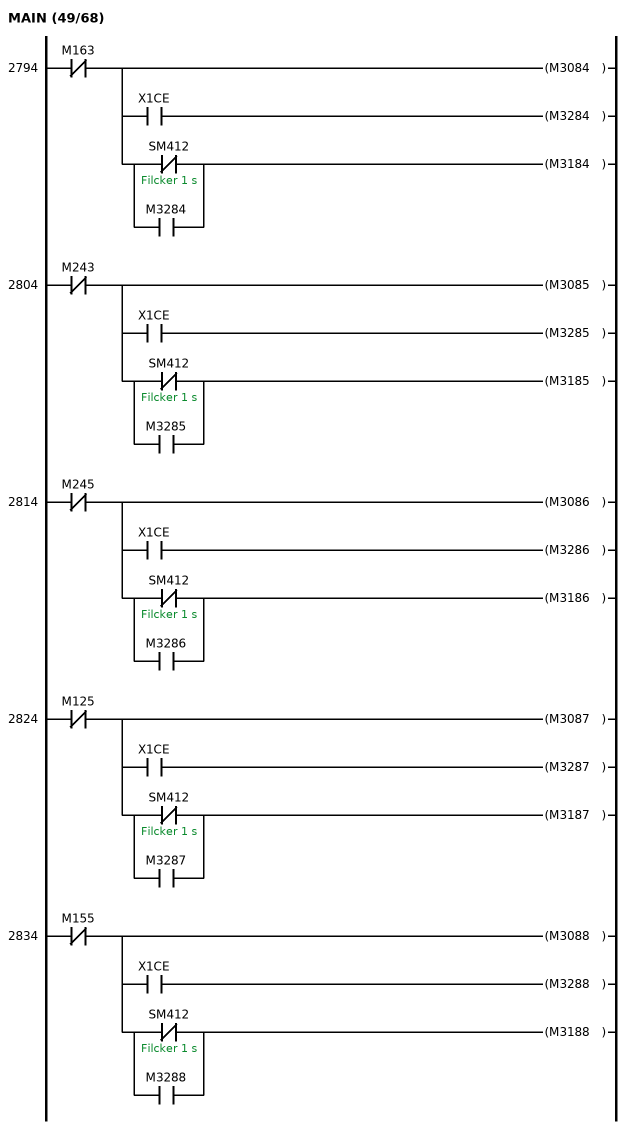
[picture p48: ladder of MAIN, rungs at steps 2794 to 2834]
2794  LDI     M163
      OUT     M3084
      MPS
      AND     X1CE
      OUT     M3284
      MPP
      LDI     SM412  ; Filcker 1 s
      OR      M3284
      ANB
      OUT     M3184
2804  LDI     M243
      OUT     M3085
      MPS
      AND     X1CE
      OUT     M3285
      MPP
      LDI     SM412  ; Filcker 1 s
      OR      M3285
      ANB
      OUT     M3185
2814  LDI     M245
      OUT     M3086
      MPS
      AND     X1CE
      OUT     M3286
      MPP
      LDI     SM412  ; Filcker 1 s
      OR      M3286
      ANB
      OUT     M3186
2824  LDI     M125
      OUT     M3087
      MPS
      AND     X1CE
      OUT     M3287
      MPP
      LDI     SM412  ; Filcker 1 s
      OR      M3287
      ANB
      OUT     M3187
2834  LDI     M155
      OUT     M3088
      MPS
      AND     X1CE
      OUT     M3288
      MPP
      LDI     SM412  ; Filcker 1 s
      OR      M3288
      ANB
      OUT     M3188
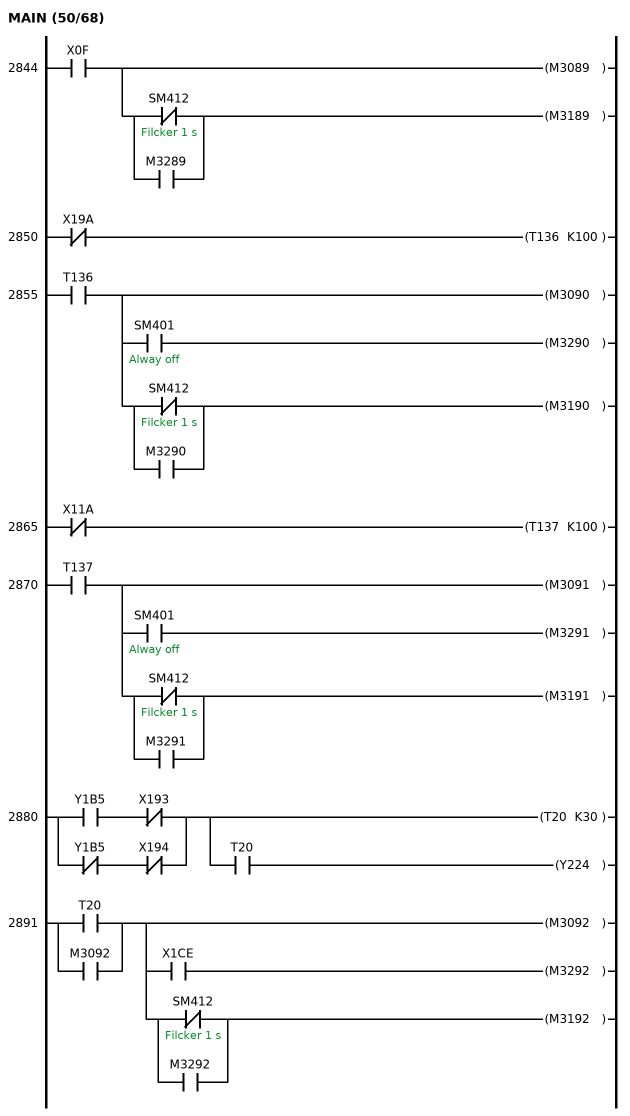
2844  LD      X0F
      OUT     M3089
      LDI     SM412  ; Filcker 1 s
      OR      M3289
      ANB
      OUT     M3189
2850  LDI     X19A
      OUT     T136 K100
2855  LD      T136
      OUT     M3090
      MPS
      AND     SM401  ; Alway off
      OUT     M3290
      MPP
      LDI     SM412  ; Filcker 1 s
      OR      M3290
      ANB
      OUT     M3190
2865  LDI     X11A
      OUT     T137 K100
2870  LD      T137
      OUT     M3091
      MPS
      AND     SM401  ; Alway off
      OUT     M3291
      MPP
      LDI     SM412  ; Filcker 1 s
      OR      M3291
      ANB
      OUT     M3191
2880  LD      Y1B5
      ANI     X193
      LDI     Y1B5
      ANI     X194
      ORB
      OUT     T20 K30
      AND     T20
      OUT     Y224
2891  LD      T20
      OR      M3092
      OUT     M3092
      MPS
      AND     X1CE
      OUT     M3292
      MPP
      LDI     SM412  ; Filcker 1 s
      OR      M3292
      ANB
      OUT     M3192
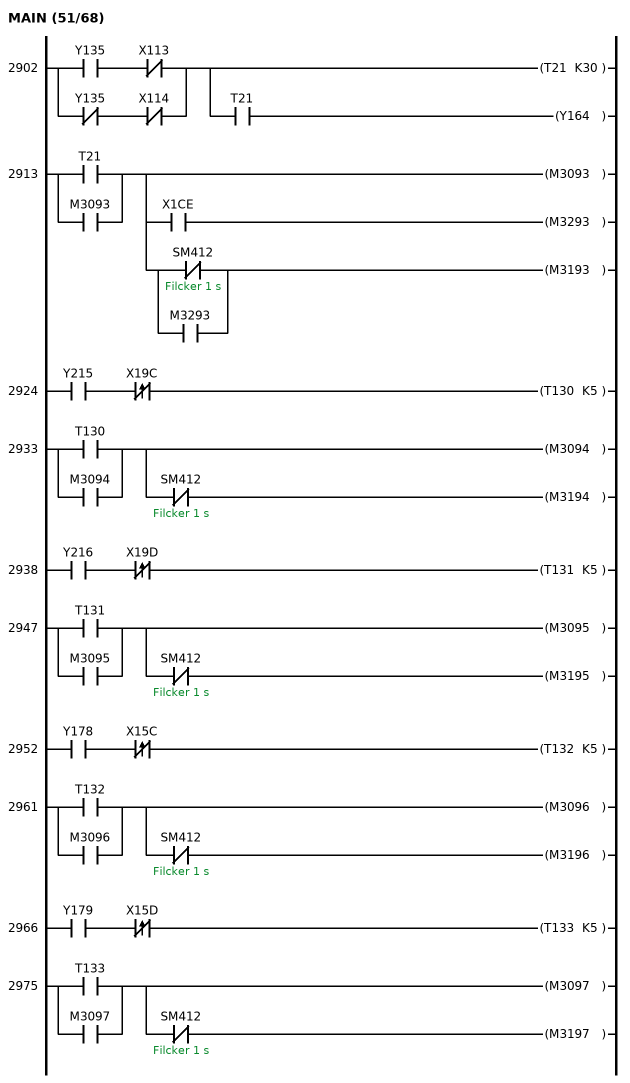
2902  LD      Y135
      ANI     X113
      LDI     Y135
      ANI     X114
      ORB
      OUT     T21 K30
      AND     T21
      OUT     Y164
2913  LD      T21
      OR      M3093
      OUT     M3093
      MPS
      AND     X1CE
      OUT     M3293
      MPP
      LDI     SM412  ; Filcker 1 s
      OR      M3293
      ANB
      OUT     M3193
2924  LD      Y215
      ANDPI   X19C
      OUT     T130 K5
2933  LD      T130
      OR      M3094
      OUT     M3094
      ANI     SM412  ; Filcker 1 s
      OUT     M3194
2938  LD      Y216
      ANDPI   X19D
      OUT     T131 K5
2947  LD      T131
      OR      M3095
      OUT     M3095
      ANI     SM412  ; Filcker 1 s
      OUT     M3195
2952  LD      Y178
      ANDPI   X15C
      OUT     T132 K5
2961  LD      T132
      OR      M3096
      OUT     M3096
      ANI     SM412  ; Filcker 1 s
      OUT     M3196
2966  LD      Y179
      ANDPI   X15D
      OUT     T133 K5
2975  LD      T133
      OR      M3097
      OUT     M3097
      ANI     SM412  ; Filcker 1 s
      OUT     M3197
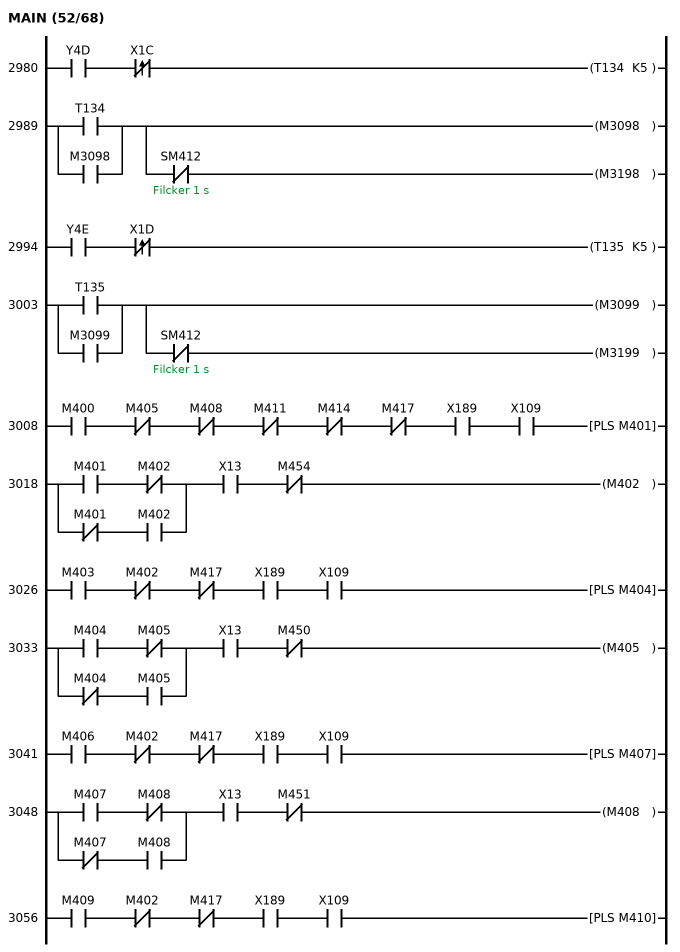
2980  LD      Y4D
      ANDPI   X1C
      OUT     T134 K5
2989  LD      T134
      OR      M3098
      OUT     M3098
      ANI     SM412  ; Filcker 1 s
      OUT     M3198
2994  LD      Y4E
      ANDPI   X1D
      OUT     T135 K5
3003  LD      T135
      OR      M3099
      OUT     M3099
      ANI     SM412  ; Filcker 1 s
      OUT     M3199
3008  LD      M400
      ANI     M405
      ANI     M408
      ANI     M411
      ANI     M414
      ANI     M417
      AND     X189
      AND     X109
      PLS     M401
3018  LD      M401
      ANI     M402
      LDI     M401
      AND     M402
      ORB
      AND     X13
      ANI     M454
      OUT     M402
3026  LD      M403
      ANI     M402
      ANI     M417
      AND     X189
      AND     X109
      PLS     M404
3033  LD      M404
      ANI     M405
      LDI     M404
      AND     M405
      ORB
      AND     X13
      ANI     M450
      OUT     M405
3041  LD      M406
      ANI     M402
      ANI     M417
      AND     X189
      AND     X109
      PLS     M407
3048  LD      M407
      ANI     M408
      LDI     M407
      AND     M408
      ORB
      AND     X13
      ANI     M451
      OUT     M408
3056  LD      M409
      ANI     M402
      ANI     M417
      AND     X189
      AND     X109
      PLS     M410
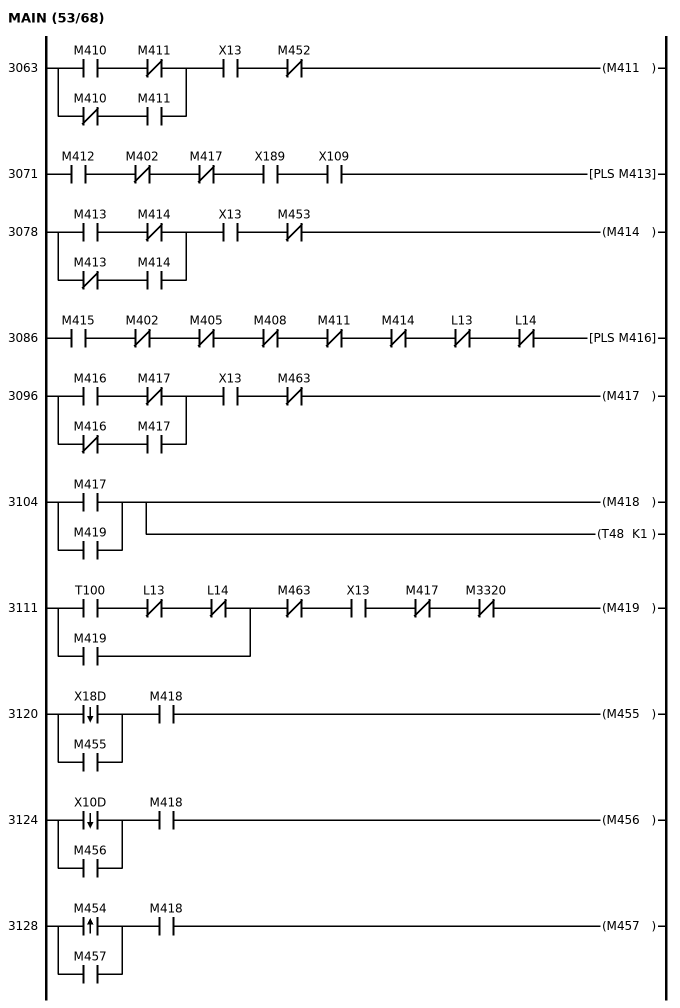
3063  LD      M410
      ANI     M411
      LDI     M410
      AND     M411
      ORB
      AND     X13
      ANI     M452
      OUT     M411
3071  LD      M412
      ANI     M402
      ANI     M417
      AND     X189
      AND     X109
      PLS     M413
3078  LD      M413
      ANI     M414
      LDI     M413
      AND     M414
      ORB
      AND     X13
      ANI     M453
      OUT     M414
3086  LD      M415
      ANI     M402
      ANI     M405
      ANI     M408
      ANI     M411
      ANI     M414
      ANI     L13
      ANI     L14
      PLS     M416
3096  LD      M416
      ANI     M417
      LDI     M416
      AND     M417
      ORB
      AND     X13
      ANI     M463
      OUT     M417
3104  LD      M417
      OR      M419
      OUT     M418
      OUT     T48 K1
3111  LD      T100
      ANI     L13
      ANI     L14
      OR      M419
      ANI     M463
      AND     X13
      ANI     M417
      ANI     M3320
      OUT     M419
3120  LDF     X18D
      OR      M455
      AND     M418
      OUT     M455
3124  LDF     X10D
      OR      M456
      AND     M418
      OUT     M456
3128  LDP     M454
      OR      M457
      AND     M418
      OUT     M457
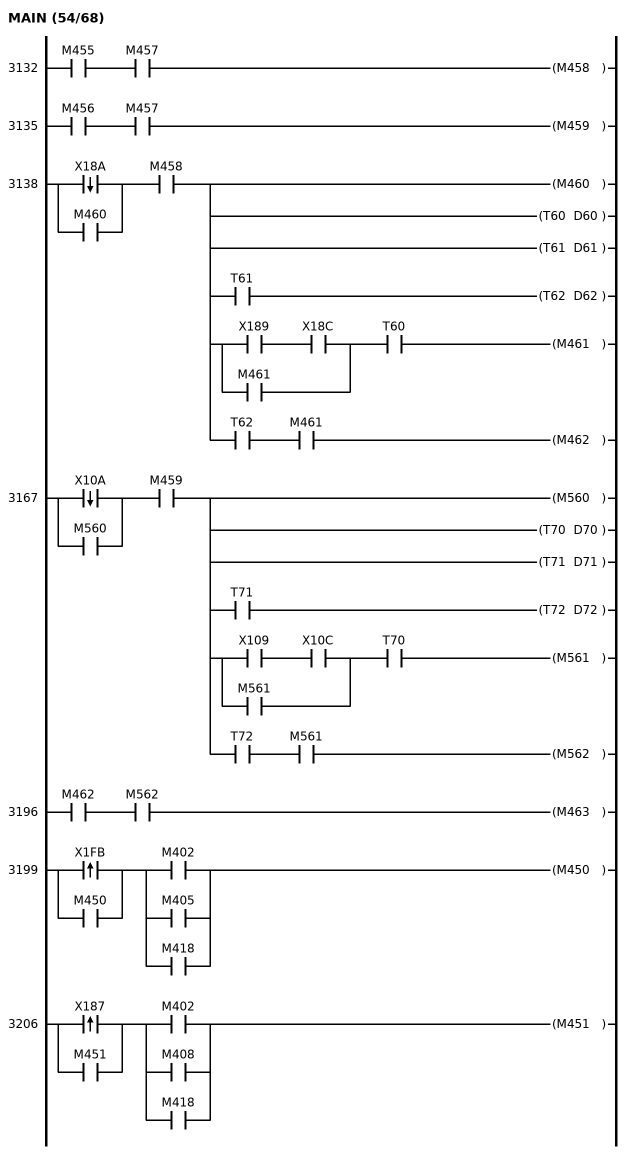
3132  LD      M455
      AND     M457
      OUT     M458
3135  LD      M456
      AND     M457
      OUT     M459
3138  LDF     X18A
      OR      M460
      AND     M458
      OUT     M460
      OUT     T60 D60
      OUT     T61 D61
      MPS
      AND     T61
      OUT     T62 D62
      MRD
      LD      X189
      AND     X18C
      OR      M461
      ANB
      AND     T60
      OUT     M461
      MPP
      AND     T62
      AND     M461
      OUT     M462
3167  LDF     X10A
      OR      M560
      AND     M459
      OUT     M560
      OUT     T70 D70
      OUT     T71 D71
      MPS
      AND     T71
      OUT     T72 D72
      MRD
      LD      X109
      AND     X10C
      OR      M561
      ANB
      AND     T70
      OUT     M561
      MPP
      AND     T72
      AND     M561
      OUT     M562
3196  LD      M462
      AND     M562
      OUT     M463
3199  LDP     X1FB
      OR      M450
      LD      M402
      OR      M405
      OR      M418
      ANB
      OUT     M450
3206  LDP     X187
      OR      M451
      LD      M402
      OR      M408
      OR      M418
      ANB
      OUT     M451
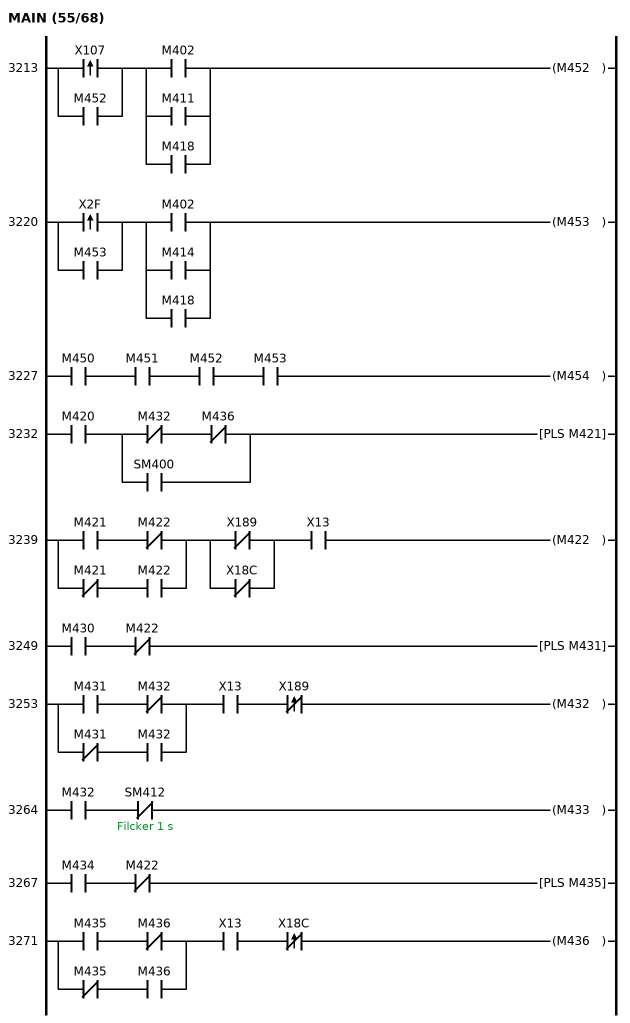
3213  LDP     X107
      OR      M452
      LD      M402
      OR      M411
      OR      M418
      ANB
      OUT     M452
3220  LDP     X2F
      OR      M453
      LD      M402
      OR      M414
      OR      M418
      ANB
      OUT     M453
3227  LD      M450
      AND     M451
      AND     M452
      AND     M453
      OUT     M454
3232  LD      M420
      LDI     M432
      ANI     M436
      OR      SM400
      ANB
      PLS     M421
3239  LD      M421
      ANI     M422
      LDI     M421
      AND     M422
      ORB
      LDI     X189
      ORI     X18C
      ANB
      AND     X13
      OUT     M422
3249  LD      M430
      ANI     M422
      PLS     M431
3253  LD      M431
      ANI     M432
      LDI     M431
      AND     M432
      ORB
      AND     X13
      ANDPI   X189
      OUT     M432
3264  LD      M432
      ANI     SM412  ; Filcker 1 s
      OUT     M433
3267  LD      M434
      ANI     M422
      PLS     M435
3271  LD      M435
      ANI     M436
      LDI     M435
      AND     M436
      ORB
      AND     X13
      ANDPI   X18C
      OUT     M436
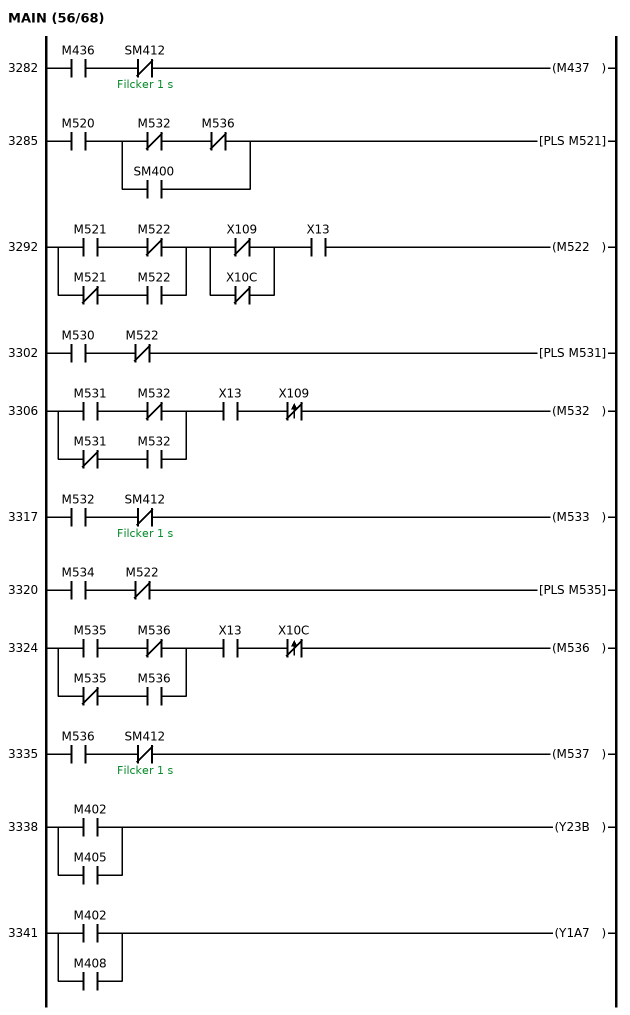
3282  LD      M436
      ANI     SM412  ; Filcker 1 s
      OUT     M437
3285  LD      M520
      LDI     M532
      ANI     M536
      OR      SM400
      ANB
      PLS     M521
3292  LD      M521
      ANI     M522
      LDI     M521
      AND     M522
      ORB
      LDI     X109
      ORI     X10C
      ANB
      AND     X13
      OUT     M522
3302  LD      M530
      ANI     M522
      PLS     M531
3306  LD      M531
      ANI     M532
      LDI     M531
      AND     M532
      ORB
      AND     X13
      ANDPI   X109
      OUT     M532
3317  LD      M532
      ANI     SM412  ; Filcker 1 s
      OUT     M533
3320  LD      M534
      ANI     M522
      PLS     M535
3324  LD      M535
      ANI     M536
      LDI     M535
      AND     M536
      ORB
      AND     X13
      ANDPI   X10C
      OUT     M536
3335  LD      M536
      ANI     SM412  ; Filcker 1 s
      OUT     M537
3338  LD      M402
      OR      M405
      OUT     Y23B
3341  LD      M402
      OR      M408
      OUT     Y1A7
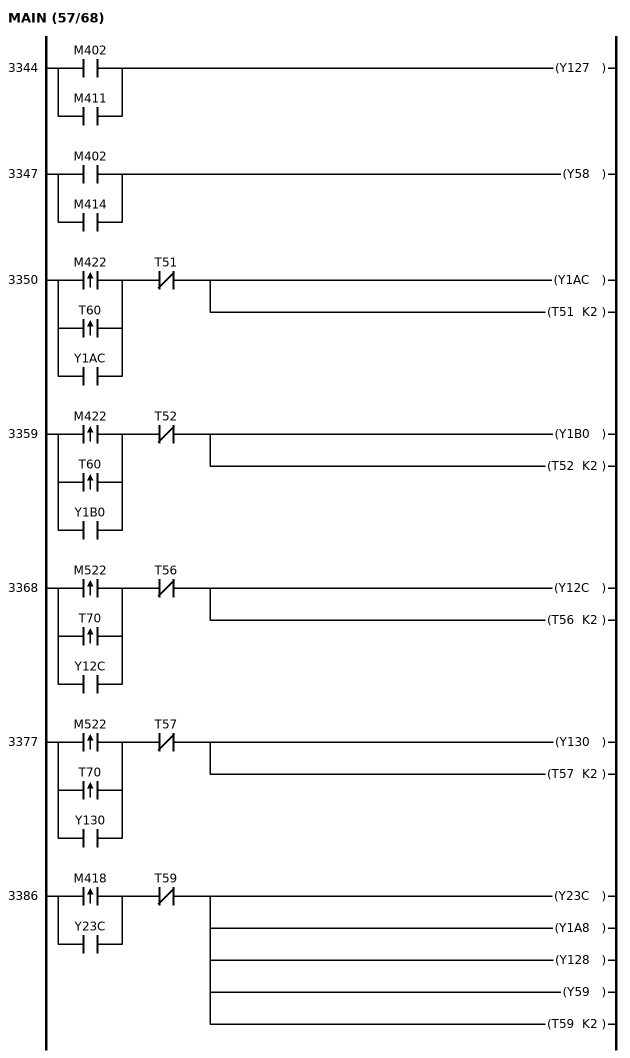
3344  LD      M402
      OR      M411
      OUT     Y127
3347  LD      M402
      OR      M414
      OUT     Y58
3350  LDP     M422
      ORP     T60
      OR      Y1AC
      ANI     T51
      OUT     Y1AC
      OUT     T51 K2
3359  LDP     M422
      ORP     T60
      OR      Y1B0
      ANI     T52
      OUT     Y1B0
      OUT     T52 K2
3368  LDP     M522
      ORP     T70
      OR      Y12C
      ANI     T56
      OUT     Y12C
      OUT     T56 K2
3377  LDP     M522
      ORP     T70
      OR      Y130
      ANI     T57
      OUT     Y130
      OUT     T57 K2
3386  LDP     M418
      OR      Y23C
      ANI     T59
      OUT     Y23C
      OUT     Y1A8
      OUT     Y128
      OUT     Y59
      OUT     T59 K2
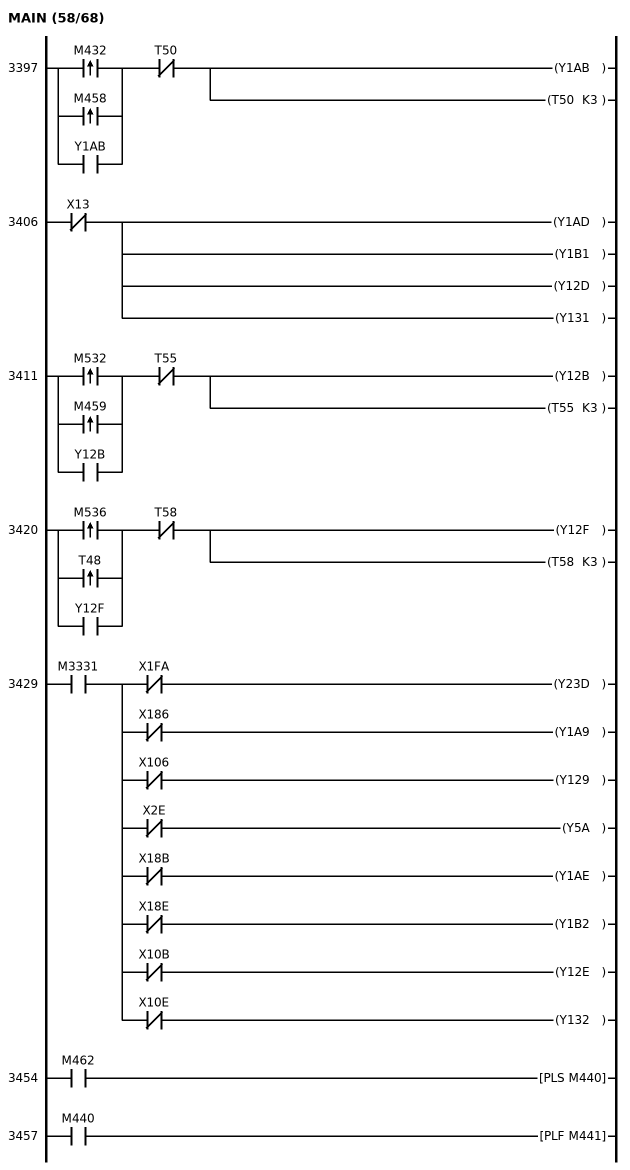
3397  LDP     M432
      ORP     M458
      OR      Y1AB
      ANI     T50
      OUT     Y1AB
      OUT     T50 K3
3406  LDI     X13
      OUT     Y1AD
      OUT     Y1B1
      OUT     Y12D
      OUT     Y131
3411  LDP     M532
      ORP     M459
      OR      Y12B
      ANI     T55
      OUT     Y12B
      OUT     T55 K3
3420  LDP     M536
      ORP     T48
      OR      Y12F
      ANI     T58
      OUT     Y12F
      OUT     T58 K3
3429  LD      M3331
      MPS
      ANI     X1FA
      OUT     Y23D
      MRD
      ANI     X186
      OUT     Y1A9
      MRD
      ANI     X106
      OUT     Y129
      MRD
      ANI     X2E
      OUT     Y5A
      MRD
      ANI     X18B
      OUT     Y1AE
      MRD
      ANI     X18E
      OUT     Y1B2
      MRD
      ANI     X10B
      OUT     Y12E
      MPP
      ANI     X10E
      OUT     Y132
3454  LD      M462
      PLS     M440
3457  LD      M440
      PLF     M441
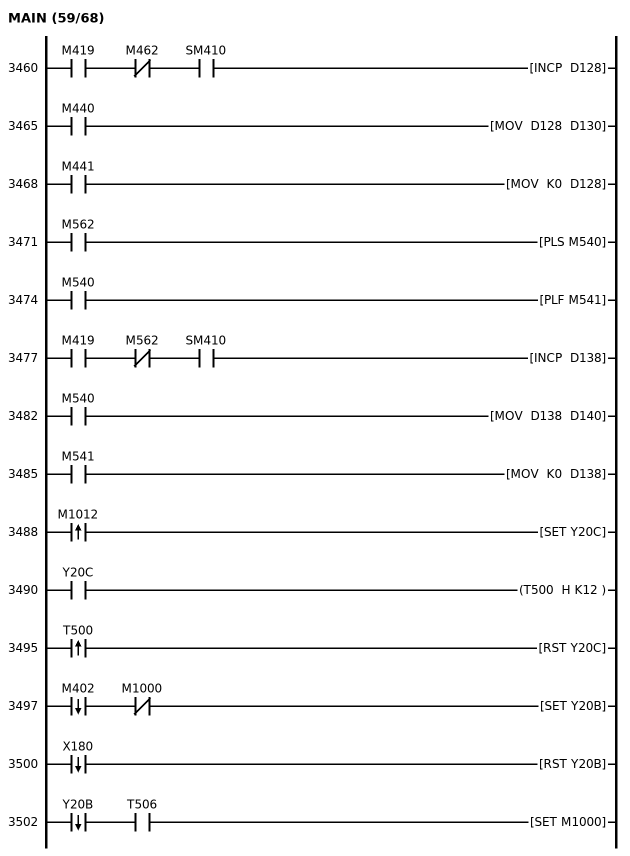
3460  LD      M419
      ANI     M462
      AND     SM410
      INCP    D128
3465  LD      M440
      MOV     D128 D130
3468  LD      M441
      MOV     K0 D128
3471  LD      M562
      PLS     M540
3474  LD      M540
      PLF     M541
3477  LD      M419
      ANI     M562
      AND     SM410
      INCP    D138
3482  LD      M540
      MOV     D138 D140
3485  LD      M541
      MOV     K0 D138
3488  LDP     M1012
      SET     Y20C
3490  LD      Y20C
      OUTH    T500 K12
3495  LDP     T500
      RST     Y20C
3497  LDF     M402
      ANI     M1000
      SET     Y20B
3500  LDF     X180
      RST     Y20B
3502  LDF     Y20B
      AND     T506
      SET     M1000
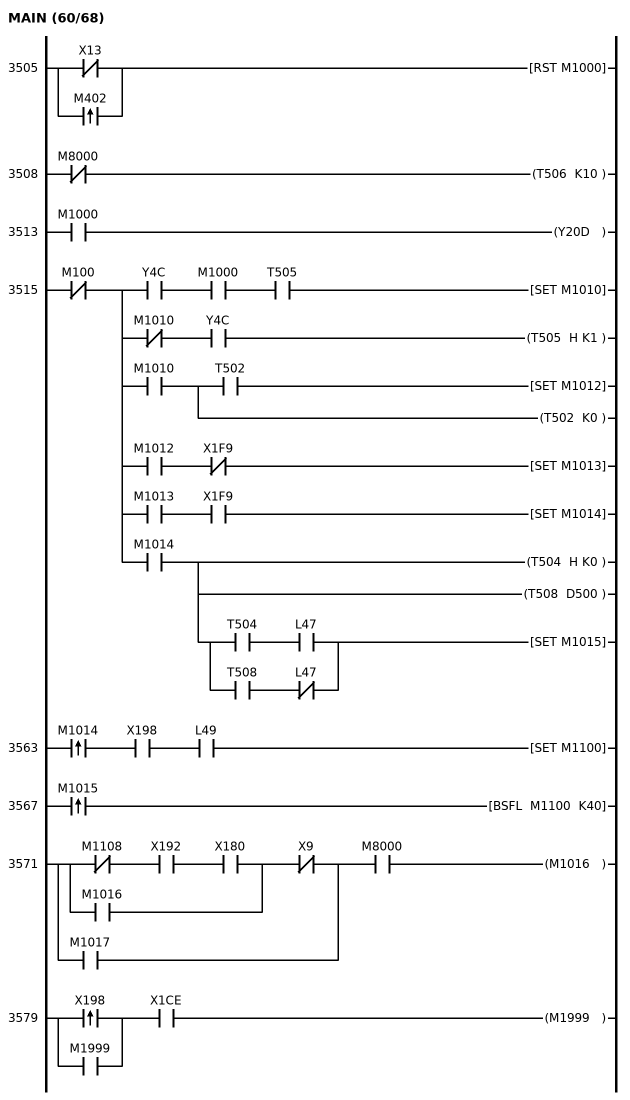
3505  LDI     X13
      ORP     M402
      RST     M1000
3508  LDI     M8000
      OUT     T506 K10
3513  LD      M1000
      OUT     Y20D
3515  LDI     M100
      MPS
      AND     Y4C
      AND     M1000
      AND     T505
      SET     M1010
      MRD
      ANI     M1010
      AND     Y4C
      OUTH    T505 K1
      MRD
      AND     M1010
      MPS
      AND     T502
      SET     M1012
      MPP
      OUT     T502 K0
      MRD
      AND     M1012
      ANI     X1F9
      SET     M1013
      MRD
      AND     M1013
      AND     X1F9
      SET     M1014
      MPP
      AND     M1014
      OUTH    T504 K0
      OUT     T508 D500
      LD      T504
      AND     L47
      LD      T508
      ANI     L47
      ORB
      ANB
      SET     M1015
3563  LDP     M1014
      AND     X198
      AND     L49
      SET     M1100
3567  LDP     M1015
      BSFL    M1100 K40
3571  LDI     M1108
      AND     X192
      AND     X180
      OR      M1016
      ANI     X9
      OR      M1017
      AND     M8000
      OUT     M1016
3579  LDP     X198
      OR      M1999
      AND     X1CE
      OUT     M1999
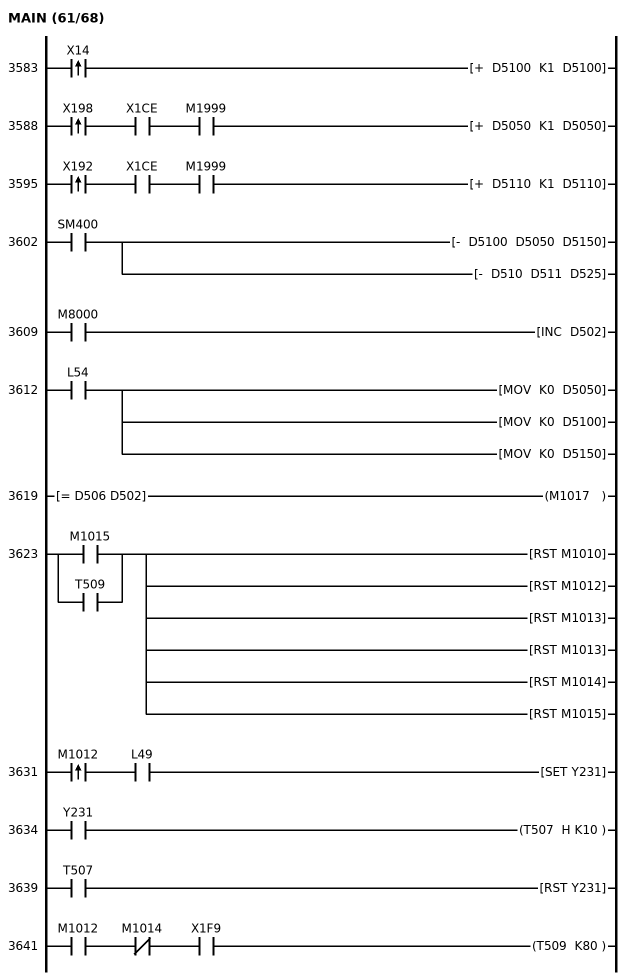
3583  LDP     X14
      +       D5100 K1 D5100
3588  LDP     X198
      AND     X1CE
      AND     M1999
      +       D5050 K1 D5050
3595  LDP     X192
      AND     X1CE
      AND     M1999
      +       D5110 K1 D5110
3602  LD      SM400
      -       D5100 D5050 D5150
      -       D510 D511 D525
3609  LD      M8000
      INC     D502
3612  LD      L54
      MOV     K0 D5050
      MOV     K0 D5100
      MOV     K0 D5150
3619  LD=     D506 D502
      OUT     M1017
3623  LD      M1015
      OR      T509
      RST     M1010
      RST     M1012
      RST     M1013
      RST     M1013
      RST     M1014
      RST     M1015
3631  LDP     M1012
      AND     L49
      SET     Y231
3634  LD      Y231
      OUTH    T507 K10
3639  LD      T507
      RST     Y231
3641  LD      M1012
      ANI     M1014
      AND     X1F9
      OUT     T509 K80
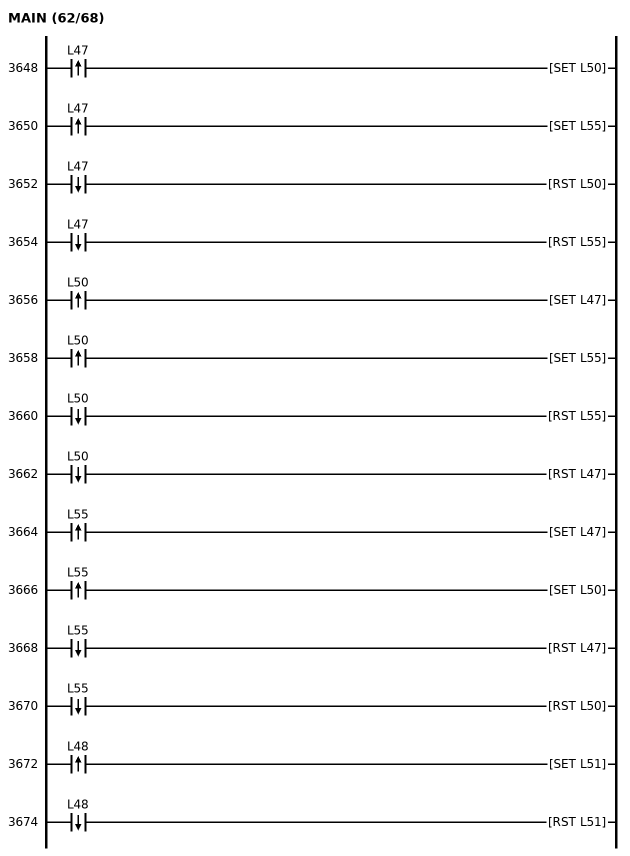
3648  LDP     L47
      SET     L50
3650  LDP     L47
      SET     L55
3652  LDF     L47
      RST     L50
3654  LDF     L47
      RST     L55
3656  LDP     L50
      SET     L47
3658  LDP     L50
      SET     L55
3660  LDF     L50
      RST     L55
3662  LDF     L50
      RST     L47
3664  LDP     L55
      SET     L47
3666  LDP     L55
      SET     L50
3668  LDF     L55
      RST     L47
3670  LDF     L55
      RST     L50
3672  LDP     L48
      SET     L51
3674  LDF     L48
      RST     L51
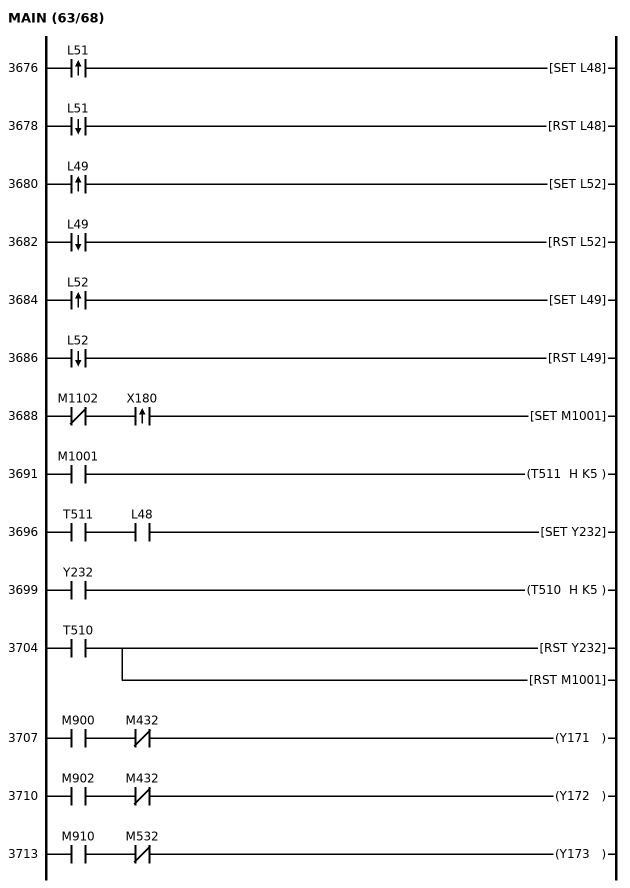
3676  LDP     L51
      SET     L48
3678  LDF     L51
      RST     L48
3680  LDP     L49
      SET     L52
3682  LDF     L49
      RST     L52
3684  LDP     L52
      SET     L49
3686  LDF     L52
      RST     L49
3688  LDI     M1102
      ANDP    X180
      SET     M1001
3691  LD      M1001
      OUTH    T511 K5
3696  LD      T511
      AND     L48
      SET     Y232
3699  LD      Y232
      OUTH    T510 K5
3704  LD      T510
      RST     Y232
      RST     M1001
3707  LD      M900
      ANI     M432
      OUT     Y171
3710  LD      M902
      ANI     M432
      OUT     Y172
3713  LD      M910
      ANI     M532
      OUT     Y173
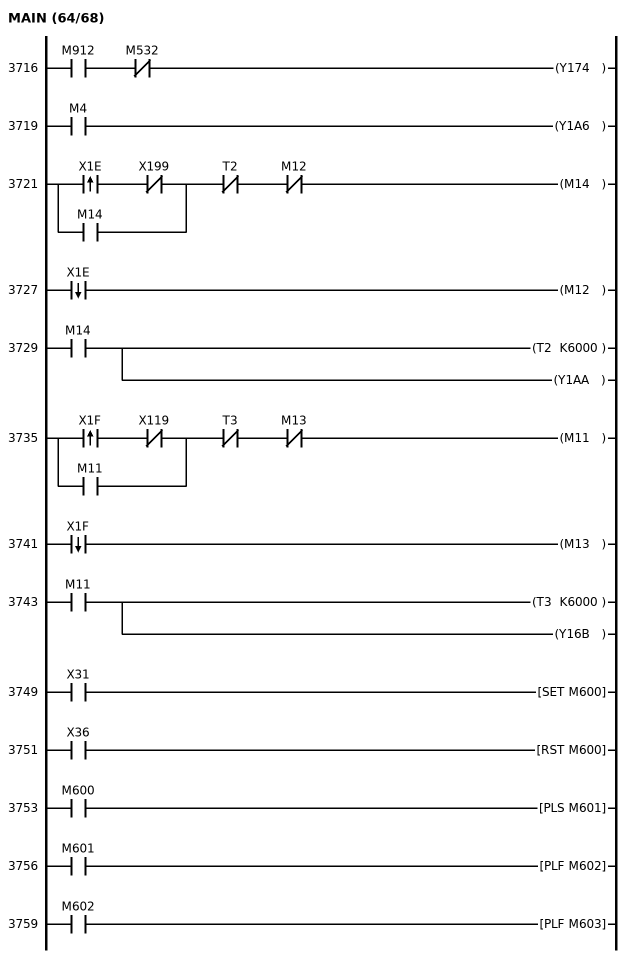
3716  LD      M912
      ANI     M532
      OUT     Y174
3719  LD      M4
      OUT     Y1A6
3721  LDP     X1E
      ANI     X199
      OR      M14
      ANI     T2
      ANI     M12
      OUT     M14
3727  LDF     X1E
      OUT     M12
3729  LD      M14
      OUT     T2 K6000
      OUT     Y1AA
3735  LDP     X1F
      ANI     X119
      OR      M11
      ANI     T3
      ANI     M13
      OUT     M11
3741  LDF     X1F
      OUT     M13
3743  LD      M11
      OUT     T3 K6000
      OUT     Y16B
3749  LD      X31
      SET     M600
3751  LD      X36
      RST     M600
3753  LD      M600
      PLS     M601
3756  LD      M601
      PLF     M602
3759  LD      M602
      PLF     M603
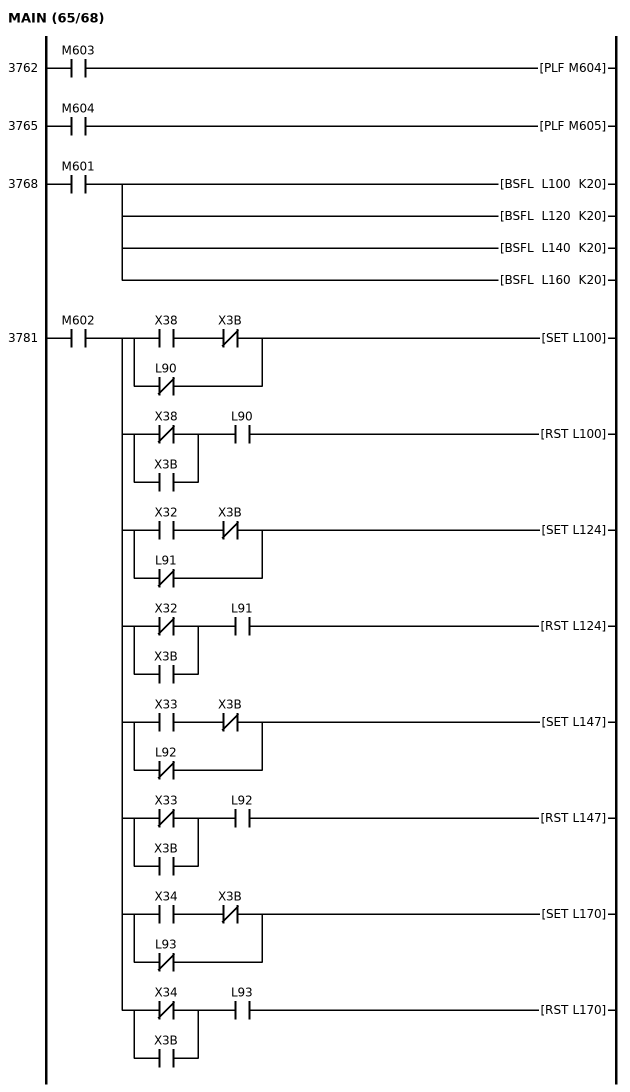
3762  LD      M603
      PLF     M604
3765  LD      M604
      PLF     M605
3768  LD      M601
      BSFL    L100 K20
      BSFL    L120 K20
      BSFL    L140 K20
      BSFL    L160 K20
3781  LD      M602
      MPS
      LD      X38
      ANI     X3B
      ORI     L90
      ANB
      SET     L100
      MRD
      LDI     X38
      OR      X3B
      ANB
      AND     L90
      RST     L100
      MRD
      LD      X32
      ANI     X3B
      ORI     L91
      ANB
      SET     L124
      MRD
      LDI     X32
      OR      X3B
      ANB
      AND     L91
      RST     L124
      MRD
      LD      X33
      ANI     X3B
      ORI     L92
      ANB
      SET     L147
      MRD
      LDI     X33
      OR      X3B
      ANB
      AND     L92
      RST     L147
      MRD
      LD      X34
      ANI     X3B
      ORI     L93
      ANB
      SET     L170
      MPP
      LDI     X34
      OR      X3B
      ANB
      AND     L93
      RST     L170
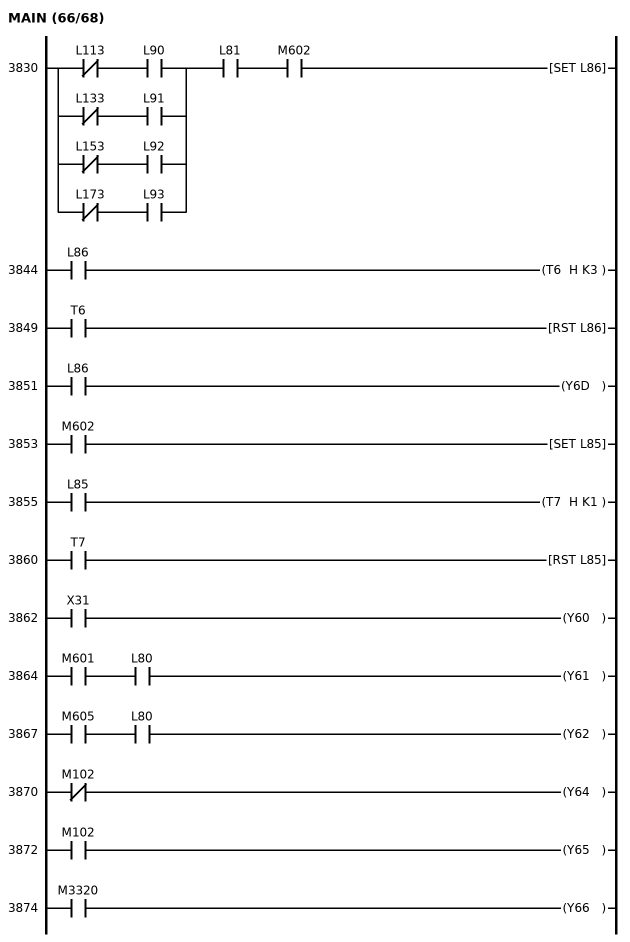
3830  LDI     L113
      AND     L90
      LDI     L133
      AND     L91
      ORB
      LDI     L153
      AND     L92
      ORB
      LDI     L173
      AND     L93
      ORB
      AND     L81
      AND     M602
      SET     L86
3844  LD      L86
      OUTH    T6 K3
3849  LD      T6
      RST     L86
3851  LD      L86
      OUT     Y6D
3853  LD      M602
      SET     L85
3855  LD      L85
      OUTH    T7 K1
3860  LD      T7
      RST     L85
3862  LD      X31
      OUT     Y60
3864  LD      M601
      AND     L80
      OUT     Y61
3867  LD      M605
      AND     L80
      OUT     Y62
3870  LDI     M102
      OUT     Y64
3872  LD      M102
      OUT     Y65
3874  LD      M3320
      OUT     Y66
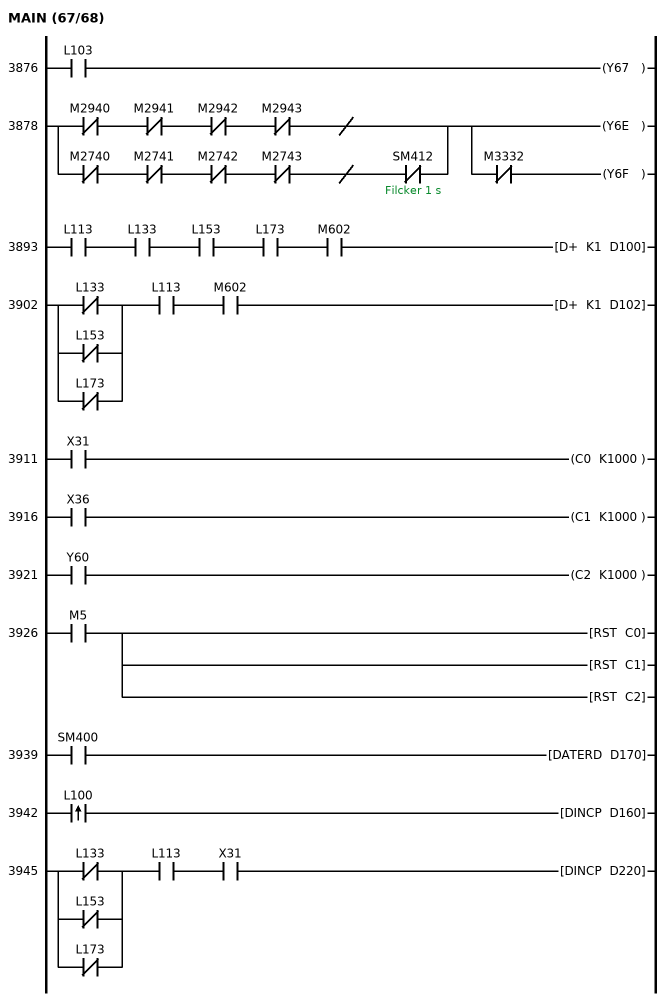
3876  LD      L103
      OUT     Y67
3878  LDI     M2940
      ANI     M2941
      ANI     M2942
      ANI     M2943
      INV
      LDI     M2740
      ANI     M2741
      ANI     M2742
      ANI     M2743
      INV
      ANI     SM412  ; Filcker 1 s
      ORB
      OUT     Y6E
      ANI     M3332
      OUT     Y6F
3893  LD      L113
      AND     L133
      AND     L153
      AND     L173
      AND     M602
      D+      K1 D100
3902  LDI     L133
      ORI     L153
      ORI     L173
      AND     L113
      AND     M602
      D+      K1 D102
3911  LD      X31
      OUT     C0 K1000
3916  LD      X36
      OUT     C1 K1000
3921  LD      Y60
      OUT     C2 K1000
3926  LD      M5
      RST     C0
      RST     C1
      RST     C2
3939  LD      SM400
      DATERD  D170
3942  LDP     L100
      DINCP   D160
3945  LDI     L133
      ORI     L153
      ORI     L173
      AND     L113
      AND     X31
      DINCP   D220
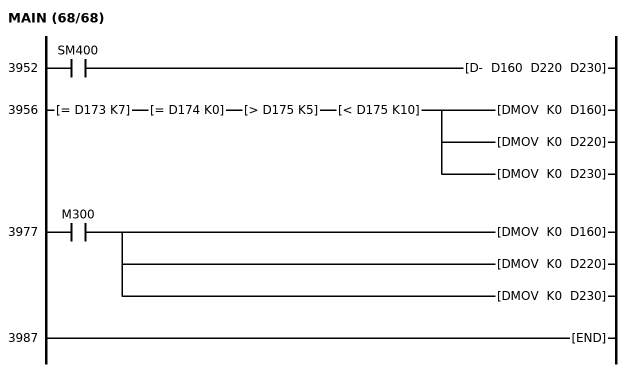
3952  LD      SM400
      D-      D160 D220 D230
3956  LD=     D173 K7
      AND=    D174 K0
      AND>    D175 K5
      AND<    D175 K10
      DMOV    K0 D160
      DMOV    K0 D220
      DMOV    K0 D230
3977  LD      M300
      DMOV    K0 D160
      DMOV    K0 D220
      DMOV    K0 D230
3987  END
END_PROGRAM

PROGRAM LOSSCODE
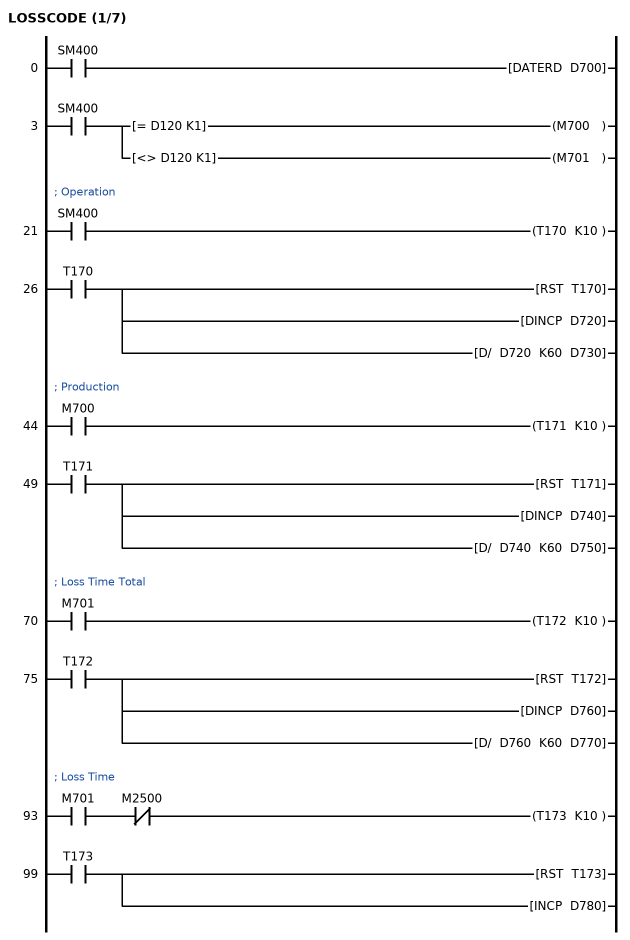
0     LD      SM400
      DATERD  D700
3     LD      SM400
      MPS
      AND=    D120 K1
      OUT     M700
      MPP
      AND<>   D120 K1
      OUT     M701
; Operation
21    LD      SM400
      OUT     T170 K10
26    LD      T170
      RST     T170
      DINCP   D720
      D/      D720 K60 D730
; Production
44    LD      M700
      OUT     T171 K10
49    LD      T171
      RST     T171
      DINCP   D740
      D/      D740 K60 D750
; Loss Time Total
70    LD      M701
      OUT     T172 K10
75    LD      T172
      RST     T172
      DINCP   D760
      D/      D760 K60 D770
; Loss Time
93    LD      M701
      ANI     M2500
      OUT     T173 K10
99    LD      T173
      RST     T173
      INCP    D780
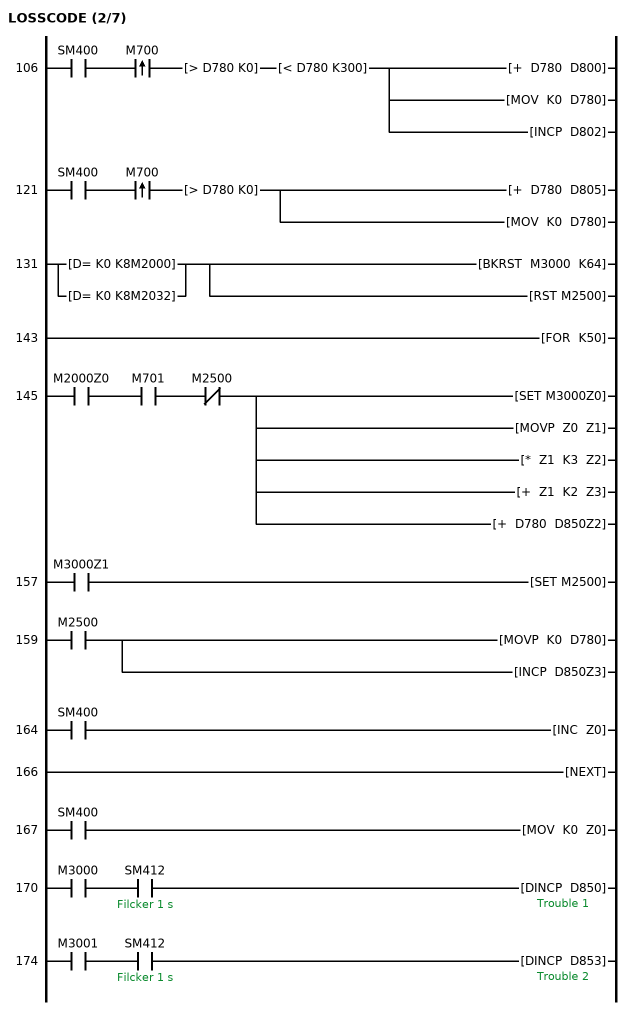
106   LD      SM400
      ANDP    M700
      AND>    D780 K0
      AND<    D780 K300
      +       D780 D800
      MOV     K0 D780
      INCP    D802
121   LD      SM400
      ANDP    M700
      AND>    D780 K0
      +       D780 D805
      MOV     K0 D780
131   LDD=    K0 K8M2000
      ORD=    K0 K8M2032
      BKRST   M3000 K64
      RST     M2500
143   FOR     K50
145   LD      M2000Z0
      AND     M701
      ANI     M2500
      SET     M3000Z0
      MOVP    Z0 Z1
      *       Z1 K3 Z2
      +       Z1 K2 Z3
      +       D780 D850Z2
157   LD      M3000Z1
      SET     M2500
159   LD      M2500
      MOVP    K0 D780
      INCP    D850Z3
164   LD      SM400
      INC     Z0
166   NEXT
167   LD      SM400
      MOV     K0 Z0
170   LD      M3000
      AND     SM412  ; Filcker 1 s
      DINCP   D850  ; Trouble 1
174   LD      M3001
      AND     SM412  ; Filcker 1 s
      DINCP   D853  ; Trouble 2
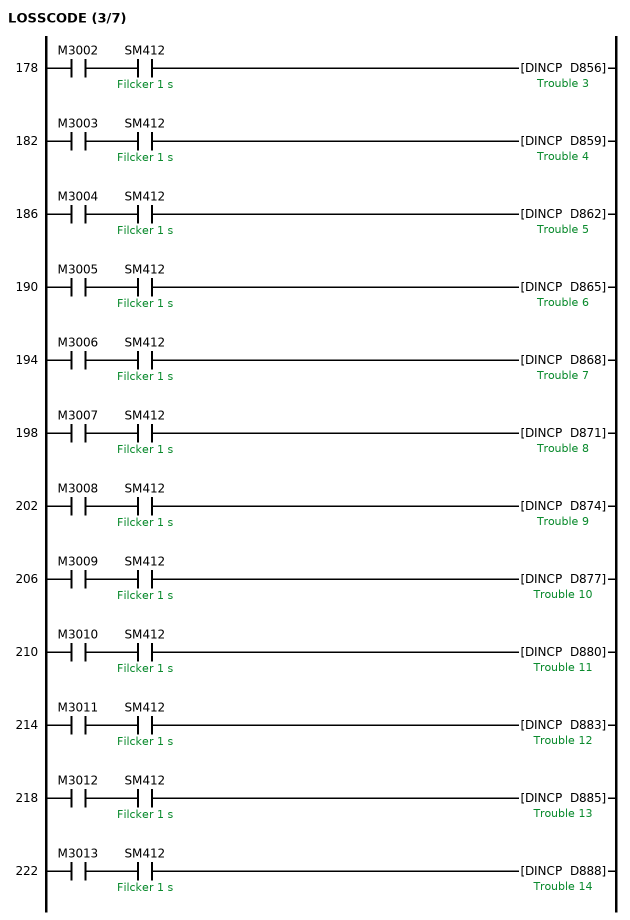
178   LD      M3002
      AND     SM412  ; Filcker 1 s
      DINCP   D856  ; Trouble 3
182   LD      M3003
      AND     SM412  ; Filcker 1 s
      DINCP   D859  ; Trouble 4
186   LD      M3004
      AND     SM412  ; Filcker 1 s
      DINCP   D862  ; Trouble 5
190   LD      M3005
      AND     SM412  ; Filcker 1 s
      DINCP   D865  ; Trouble 6
194   LD      M3006
      AND     SM412  ; Filcker 1 s
      DINCP   D868  ; Trouble 7
198   LD      M3007
      AND     SM412  ; Filcker 1 s
      DINCP   D871  ; Trouble 8
202   LD      M3008
      AND     SM412  ; Filcker 1 s
      DINCP   D874  ; Trouble 9
206   LD      M3009
      AND     SM412  ; Filcker 1 s
      DINCP   D877  ; Trouble 10
210   LD      M3010
      AND     SM412  ; Filcker 1 s
      DINCP   D880  ; Trouble 11
214   LD      M3011
      AND     SM412  ; Filcker 1 s
      DINCP   D883  ; Trouble 12
218   LD      M3012
      AND     SM412  ; Filcker 1 s
      DINCP   D885  ; Trouble 13
222   LD      M3013
      AND     SM412  ; Filcker 1 s
      DINCP   D888  ; Trouble 14
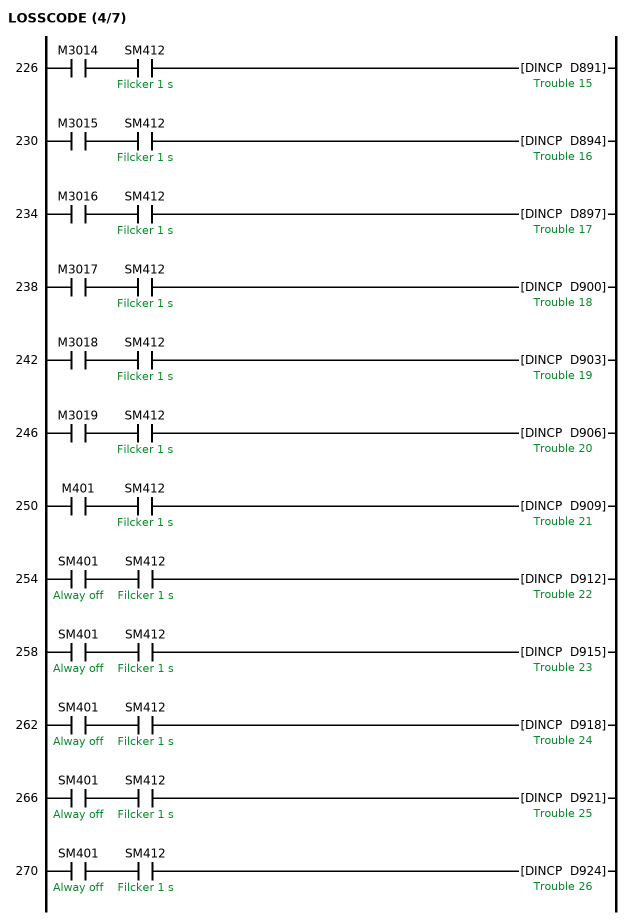
226   LD      M3014
      AND     SM412  ; Filcker 1 s
      DINCP   D891  ; Trouble 15
230   LD      M3015
      AND     SM412  ; Filcker 1 s
      DINCP   D894  ; Trouble 16
234   LD      M3016
      AND     SM412  ; Filcker 1 s
      DINCP   D897  ; Trouble 17
238   LD      M3017
      AND     SM412  ; Filcker 1 s
      DINCP   D900  ; Trouble 18
242   LD      M3018
      AND     SM412  ; Filcker 1 s
      DINCP   D903  ; Trouble 19
246   LD      M3019
      AND     SM412  ; Filcker 1 s
      DINCP   D906  ; Trouble 20
250   LD      M401
      AND     SM412  ; Filcker 1 s
      DINCP   D909  ; Trouble 21
254   LD      SM401  ; Alway off
      AND     SM412  ; Filcker 1 s
      DINCP   D912  ; Trouble 22
258   LD      SM401  ; Alway off
      AND     SM412  ; Filcker 1 s
      DINCP   D915  ; Trouble 23
262   LD      SM401  ; Alway off
      AND     SM412  ; Filcker 1 s
      DINCP   D918  ; Trouble 24
266   LD      SM401  ; Alway off
      AND     SM412  ; Filcker 1 s
      DINCP   D921  ; Trouble 25
270   LD      SM401  ; Alway off
      AND     SM412  ; Filcker 1 s
      DINCP   D924  ; Trouble 26
